// Mitsubishi GX Works2 project: hung_creat_plc   PLC: FX3U/FX3UC

PROGRAM MAIN
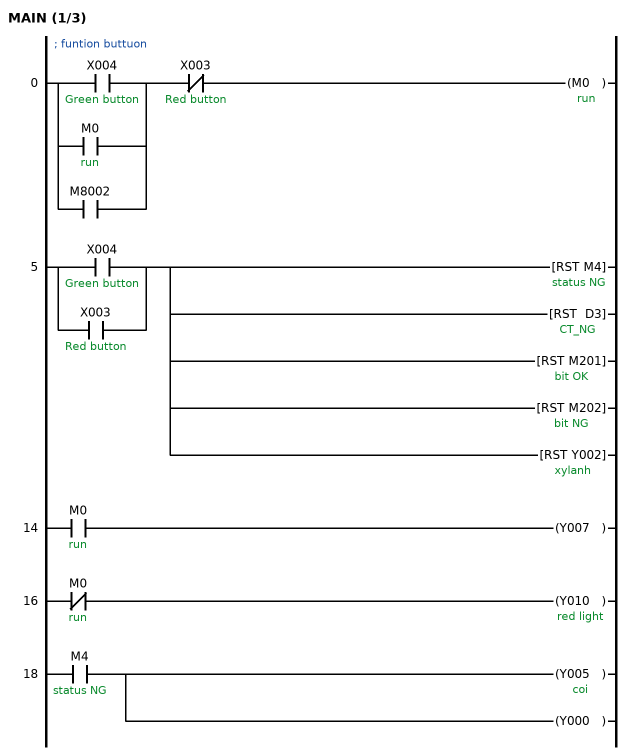
; funtion buttuon
0     LD      X004  ; Green button
      OR      M0  ; run
      OR      M8002
      ANI     X003  ; Red button
      OUT     M0  ; run
5     LD      X004  ; Green button
      OR      X003  ; Red button
      RST     M4  ; status NG
      RST     D3  ; CT_NG
      RST     M201  ; bit OK
      RST     M202  ; bit NG
      RST     Y002  ; xylanh
14    LD      M0  ; run
      OUT     Y007
16    LDI     M0  ; run
      OUT     Y010  ; red light
18    LD      M4  ; status NG
      OUT     Y005  ; coi
      OUT     Y000
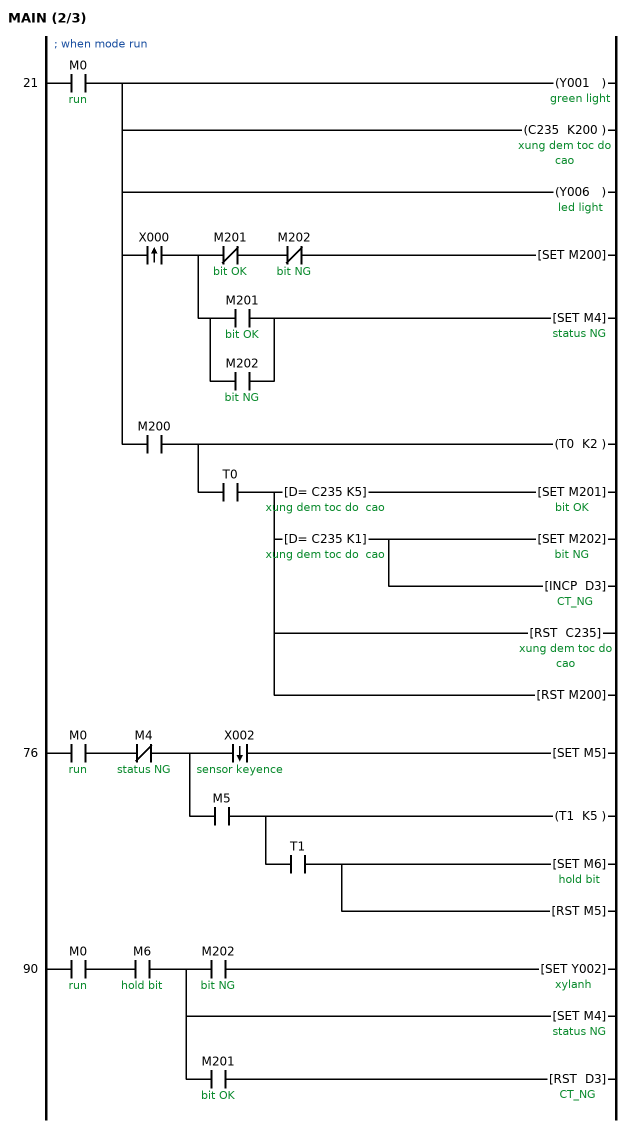
; when mode run
21    LD      M0  ; run
      OUT     Y001  ; green light
      OUT     C235 K200  ; xung dem toc do  cao
      OUT     Y006  ; led light
      MPS
      ANDP    X000
      MPS
      ANI     M201  ; bit OK
      ANI     M202  ; bit NG
      SET     M200
      MPP
      LD      M201  ; bit OK
      OR      M202  ; bit NG
      ANB
      SET     M4  ; status NG
      MPP
      AND     M200
      OUT     T0 K2
      AND     T0
      MPS
      ANDD=   C235 K5  ; xung dem toc do  cao
      SET     M201  ; bit OK
      MRD
      ANDD=   C235 K1  ; xung dem toc do  cao
      SET     M202  ; bit NG
      INCP    D3
      MPP
      RST     C235  ; xung dem toc do  cao
      RST     M200
76    LD      M0  ; run
      ANI     M4  ; status NG
      MPS
      ANDF    X002  ; sensor keyence
      SET     M5
      MPP
      AND     M5
      OUT     T1 K5
      AND     T1
      SET     M6  ; hold bit
      RST     M5
90    LD      M0  ; run
      AND     M6  ; hold bit
      MPS
      AND     M202  ; bit NG
      SET     Y002  ; xylanh
      MPP
      SET     M4  ; status NG
      AND     M201  ; bit OK
      RST     D3  ; CT_NG
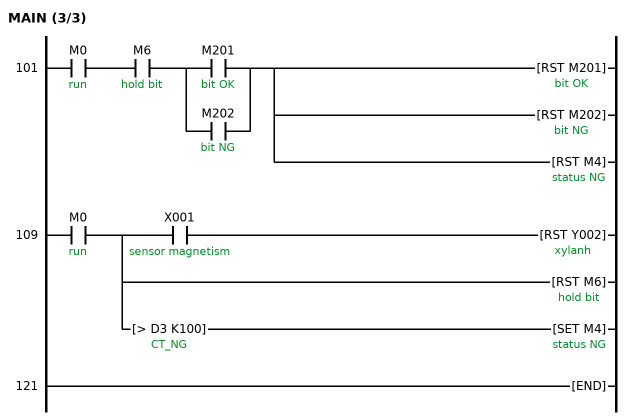
101   LD      M0  ; run
      AND     M6  ; hold bit
      LD      M201  ; bit OK
      OR      M202  ; bit NG
      ANB
      RST     M201  ; bit OK
      RST     M202  ; bit NG
      RST     M4  ; status NG
109   LD      M0  ; run
      MPS
      AND     X001  ; sensor magnetism
      RST     Y002  ; xylanh
      MPP
      RST     M6  ; hold bit
      AND>    D3 K100  ; CT_NG
      SET     M4  ; status NG
121   END
END_PROGRAM

// device comments not shown above
D0  ; CT
M3  ; bit reset NG and OK
